% RSLogix 500 project TRAFFIC LIGHT.RSS, saved by version 8.30.00.16 %
PROJECT "UNTITLED"    % processor: Bul.1763 MicroLogix 1100 Series B %

PROGRAM FILES
  LAD 2   7 rungs

DATA FILES
  O0 OUTPUT  4 elements
  I1 INPUT  6 elements
  S2 STATUS  66 elements
  B3 BINARY  1 elements
  T4 TIMER  1 elements
  C5 COUNTER  1 elements
  R6 CONTROL  1 elements
  N7 INTEGER  1 elements
  F8 FLOAT  1 elements

LADDER 2
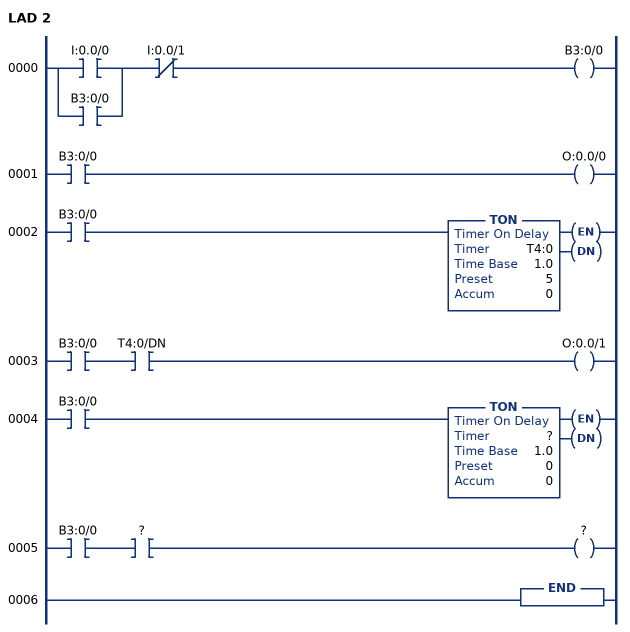
% Rung: 0 %  % edit flag set %
SOR BST XIC I:0.0/0 NXB XIC B3:0/0 BND XIO I:0.0/1 OTE B3:0/0 EOR
% Rung: 1 %  % edit flag set %
SOR XIC B3:0/0 OTE O:0.0/0 EOR
% Rung: 2 %  % edit flag set %
SOR XIC B3:0/0 TON T4:0 1.0 5 0 EOR
% Rung: 3 %  % edit flag set %
SOR XIC B3:0/0 XIC T4:0/DN OTE O:0.0/1 EOR
% Rung: 4 %  % edit flag set %
SOR XIC B3:0/0 TON ? 1.0 0 0 EOR
% Rung: 5 %  % edit flag set %
SOR XIC B3:0/0 XIC ? OTE ? EOR
% Rung: 6 %
SOR END EOR
